FUNCTION_BLOCK FB_SortingByWeight
VAR_INPUT
END_VAR
VAR_OUTPUT
END_VAR
VAR
	WeighingDone : BOOL;
	dummy : BOOL;
END_VAR
VAR_IN_OUT
	control_data : PlantAndCMs.Udt_PlantControl_Mode_1;
	
END_VAR

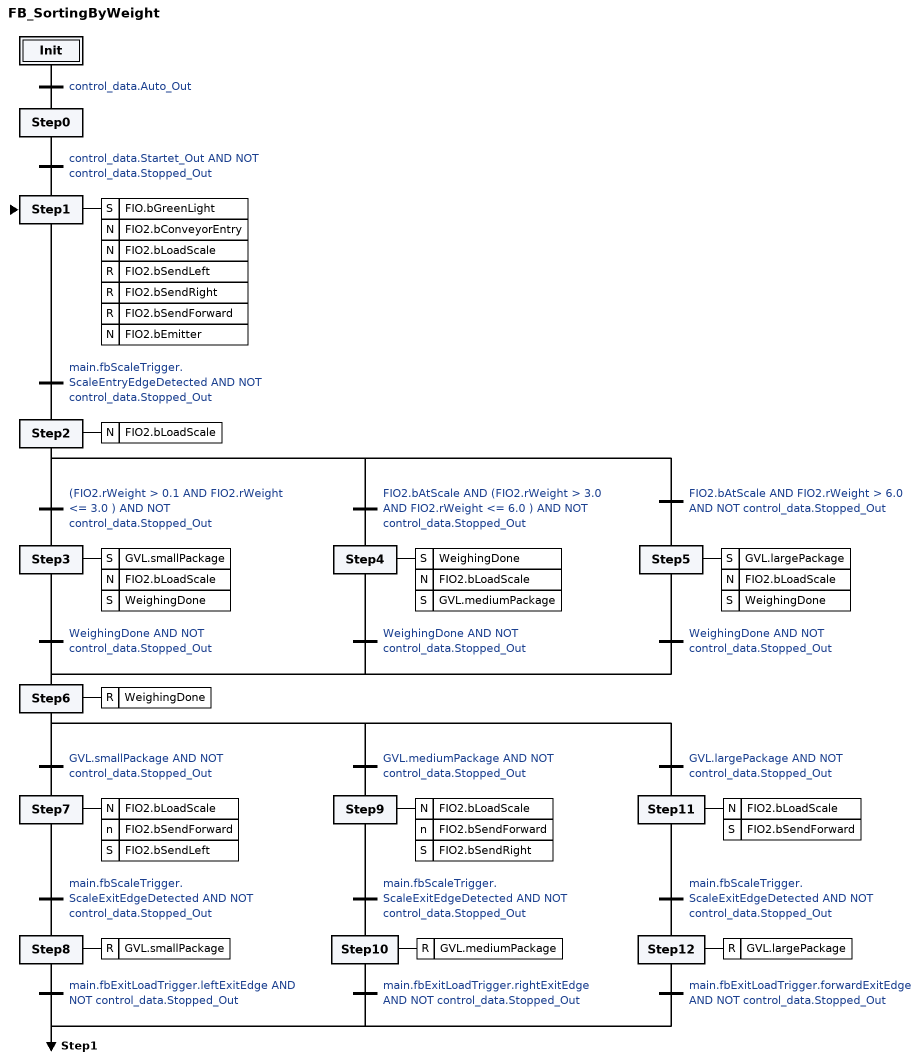
INITIAL_STEP Init:
END_STEP
TRANSITION FROM Init TO Step0
    := control_data.Auto_Out;
END_TRANSITION
STEP Step0:
END_STEP
TRANSITION FROM Step0 TO Step1
    := control_data.Startet_Out AND NOT control_data.Stopped_Out;
END_TRANSITION
STEP Step1:
    FIO.bGreenLight(S);
    FIO2.bConveyorEntry(N);
    FIO2.bLoadScale(N);
    FIO2.bSendLeft(R);
    FIO2.bSendRight(R);
    FIO2.bSendForward(R);
    FIO2.bEmitter(N);
END_STEP
TRANSITION FROM Step1 TO Step2
    := main.fbScaleTrigger.ScaleEntryEdgeDetected AND NOT control_data.Stopped_Out;
END_TRANSITION
STEP Step2:
    FIO2.bLoadScale(N);
END_STEP
TRANSITION FROM Step2 TO Step3
    := (FIO2.rWeight > 0.1 AND FIO2.rWeight <= 3.0 ) AND NOT control_data.Stopped_Out;
END_TRANSITION
STEP Step3:
    GVL.smallPackage(S);
    FIO2.bLoadScale(N);
    WeighingDone(S);
END_STEP
TRANSITION FROM Step3 TO Step6
    := WeighingDone AND NOT control_data.Stopped_Out;
END_TRANSITION
TRANSITION FROM Step2 TO Step4
    := FIO2.bAtScale AND (FIO2.rWeight > 3.0 AND FIO2.rWeight <= 6.0 ) AND NOT control_data.Stopped_Out;
END_TRANSITION
STEP Step4:
    WeighingDone(S);
    FIO2.bLoadScale(N);
    GVL.mediumPackage(S);
END_STEP
TRANSITION FROM Step4 TO Step6
    := WeighingDone AND NOT control_data.Stopped_Out;
END_TRANSITION
TRANSITION FROM Step2 TO Step5
    := FIO2.bAtScale AND FIO2.rWeight > 6.0 AND NOT control_data.Stopped_Out;
END_TRANSITION
STEP Step5:
    GVL.largePackage(S);
    FIO2.bLoadScale(N);
    WeighingDone(S);
END_STEP
TRANSITION FROM Step5 TO Step6
    := WeighingDone AND NOT control_data.Stopped_Out;
END_TRANSITION
STEP Step6:
    WeighingDone(R);
END_STEP
TRANSITION FROM Step6 TO Step7
    := GVL.smallPackage AND NOT control_data.Stopped_Out;
END_TRANSITION
STEP Step7:
    FIO2.bLoadScale(N);
    FIO2.bSendForward(n);
    FIO2.bSendLeft(S);
END_STEP
TRANSITION FROM Step7 TO Step8
    := main.fbScaleTrigger.ScaleExitEdgeDetected AND NOT control_data.Stopped_Out;
END_TRANSITION
STEP Step8:
    GVL.smallPackage(R);
END_STEP
TRANSITION FROM Step8 TO Step1
    := main.fbExitLoadTrigger.leftExitEdge AND NOT control_data.Stopped_Out;
END_TRANSITION
TRANSITION FROM Step6 TO Step9
    := GVL.mediumPackage AND NOT control_data.Stopped_Out;
END_TRANSITION
STEP Step9:
    FIO2.bLoadScale(N);
    FIO2.bSendForward(n);
    FIO2.bSendRight(S);
END_STEP
TRANSITION FROM Step9 TO Step10
    := main.fbScaleTrigger.ScaleExitEdgeDetected AND NOT control_data.Stopped_Out;
END_TRANSITION
STEP Step10:
    GVL.mediumPackage(R);
END_STEP
TRANSITION FROM Step10 TO Step1
    := main.fbExitLoadTrigger.rightExitEdge AND NOT control_data.Stopped_Out;
END_TRANSITION
TRANSITION FROM Step6 TO Step11
    := GVL.largePackage AND NOT control_data.Stopped_Out;
END_TRANSITION
STEP Step11:
    FIO2.bLoadScale(N);
    FIO2.bSendForward(S);
END_STEP
TRANSITION FROM Step11 TO Step12
    := main.fbScaleTrigger.ScaleExitEdgeDetected AND NOT control_data.Stopped_Out;
END_TRANSITION
STEP Step12:
    GVL.largePackage(R);
END_STEP
TRANSITION FROM Step12 TO Step1
    := main.fbExitLoadTrigger.forwardExitEdge AND NOT control_data.Stopped_Out;
END_TRANSITION

END_FUNCTION_BLOCK

(* stored: Version 1.1.0.1, ProductVersion 3.1.4024.13
   POU FB_SortingByWeight: Id {09a00958-a6c7-4482-950f-f9586603509a}, SpecialFunc None *)
